// Mitsubishi GX Works2 project: intel   PLC: Q03UDV

PROGRAM MAIN
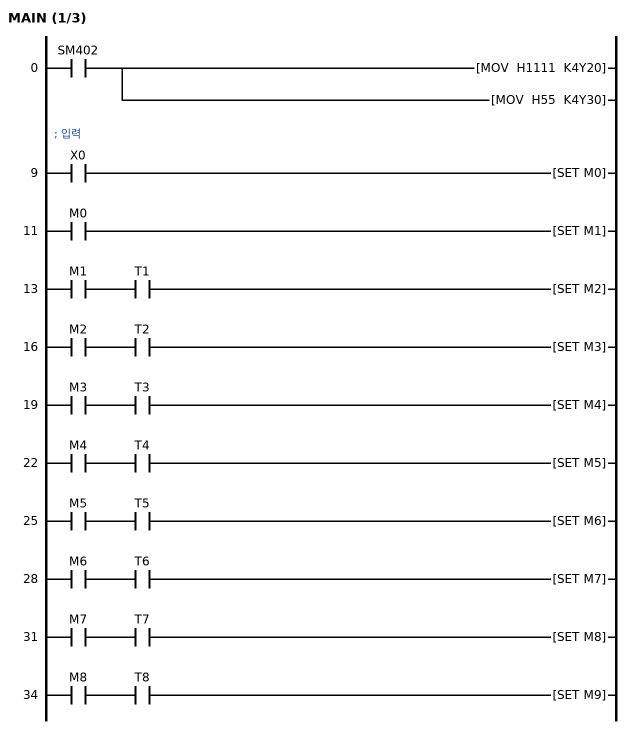
0     LD      SM402
      MOV     H1111 K4Y20
      MOV     H55 K4Y30
; 입력
9     LD      X0
      SET     M0
11    LD      M0
      SET     M1
13    LD      M1
      AND     T1
      SET     M2
16    LD      M2
      AND     T2
      SET     M3
19    LD      M3
      AND     T3
      SET     M4
22    LD      M4
      AND     T4
      SET     M5
25    LD      M5
      AND     T5
      SET     M6
28    LD      M6
      AND     T6
      SET     M7
31    LD      M7
      AND     T7
      SET     M8
34    LD      M8
      AND     T8
      SET     M9
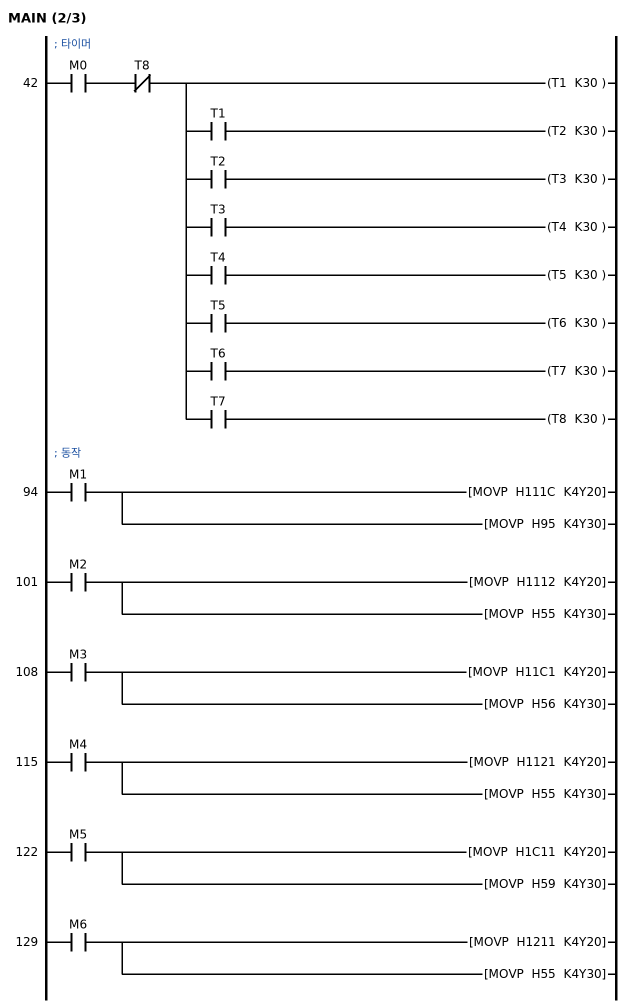
; 타이머
42    LD      M0
      ANI     T8
      OUT     T1 K30
      MPS
      AND     T1
      OUT     T2 K30
      MRD
      AND     T2
      OUT     T3 K30
      MRD
      AND     T3
      OUT     T4 K30
      MRD
      AND     T4
      OUT     T5 K30
      MRD
      AND     T5
      OUT     T6 K30
      MRD
      AND     T6
      OUT     T7 K30
      MPP
      AND     T7
      OUT     T8 K30
; 동작
94    LD      M1
      MOVP    H111C K4Y20
      MOVP    H95 K4Y30
101   LD      M2
      MOVP    H1112 K4Y20
      MOVP    H55 K4Y30
108   LD      M3
      MOVP    H11C1 K4Y20
      MOVP    H56 K4Y30
115   LD      M4
      MOVP    H1121 K4Y20
      MOVP    H55 K4Y30
122   LD      M5
      MOVP    H1C11 K4Y20
      MOVP    H59 K4Y30
129   LD      M6
      MOVP    H1211 K4Y20
      MOVP    H55 K4Y30
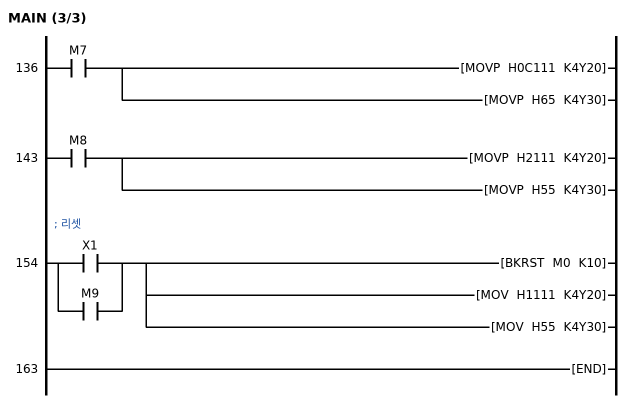
136   LD      M7
      MOVP    H0C111 K4Y20
      MOVP    H65 K4Y30
143   LD      M8
      MOVP    H2111 K4Y20
      MOVP    H55 K4Y30
; 리셋
154   LD      X1
      OR      M9
      BKRST   M0 K10
      MOV     H1111 K4Y20
      MOV     H55 K4Y30
163   END
END_PROGRAM
